FUNCTION_BLOCK FB_Pump
VAR_OUTPUT
	nPressure: REAL; // [Volts]
END_VAR
VAR
	// bRelayOn AT %Q* : BOOL := FALSE; // True = On
	bRelayOn : BOOL := FALSE;
	// nCurrentPressure AT %I* : REAL; // Volts
	bValveOpen : BOOL := FALSE;
END_VAR

// For Simulation
IF bValveOpen THEN
	GVL_VAR.bValve := TRUE;
	GVL_VAR.bPump := FALSE;
ELSIF bRelayOn THEN
	GVL_VAR.bPump := TRUE;
	GVL_VAR.bValve := FALSE;
ELSE
	GVL_VAR.bPump := FALSE;
	GVL_VAR.bValve := FALSE;
END_IF
nPressure := GVL_VAR.nPressure;

METHOD PUBLIC SetRelay : BOOL
VAR_INPUT
	bRelayState : BOOL;
END_VAR
bRelayOn := bRelayState;
SetRelay := TRUE;
END_METHOD

METHOD PUBLIC SetValve : BOOL
VAR_INPUT
	bValveState : BOOL;
END_VAR
bValveOpen := bValveState;
SetValve := TRUE;
END_METHOD

END_FUNCTION_BLOCK

(* stored: Version 1.1.0.1, ProductVersion 3.1.4024.12
   POU FB_Pump: Id {2189f6e3-949f-4eb4-811c-6a2452780df7}, SpecialFunc None
   Method SetRelay: Id {ef407a0f-9ab4-4891-b141-81e8459e209e}
   Method SetValve: Id {78bc9e55-eb77-405d-b9c0-9a18632c1385} *)
